{attribute 'GeneratedUsingTerminal: AT2041-5250-0019'}
{attribute addProperty BoxType "AT2041-5250-0019"}
{attribute addProperty Id "FB_InputsAT %I*FB_Inputs_4BC4AA0166FB_OutputsAT %Q*FB_Outputs_DAFD38E02WcStateAT %I*WcState_9091E0EB2InfoDataAT %I*InfoData_A7436BC610"}
{attribute addProperty CRC "866377499"}
{attribute addProperty Size "80"}
TYPE AT2041_33A3DF1B EXTENDS EtcSlaveTerminalBase_947E5A46 :
STRUCT
	{attribute addProperty Name "FB_Inputs"}
	FB_Inputs : FB_Inputs_4BC4AA01;
	{attribute addProperty Name "FB_Outputs"}
	FB_Outputs : FB_Outputs_DAFD38E0;
	{attribute addProperty Name "WcState"}
	WcState : WcState_9091E0EB;
	{attribute addProperty Name "InfoData"}
	InfoData : InfoData_A7436BC6;
END_STRUCT
END_TYPE
